FUNCTION_BLOCK FB_FIFO_1 EXTENDS FB_FIFO_OOP
VAR_INPUT
END_VAR
VAR_OUTPUT
END_VAR
VAR
END_VAR

PROPERTY ifEmptyRegister : IF_EmptyRegister
GET
ifEmptyRegister:=super^;
END_GET
END_PROPERTY

PROPERTY ifFillRegister : IF_FillRegister
GET
ifFillRegister:=super^;
END_GET
END_PROPERTY

PROPERTY ifRegister : IF_Register
GET
ifRegister:=super^;
END_GET
END_PROPERTY

END_FUNCTION_BLOCK

(* stored: Version 1.1.0.1
   POU FB_FIFO_1: Id {7d20f1f5-68f8-4dda-a4fa-66e225c03a6c}, SpecialFunc None
   Property ifEmptyRegister: Id {7cd02d5f-3e9f-42f9-b54d-32ee951b56ff}
   Get Get: Id {1e8b9ca5-eaab-40e5-82b7-e5efa8257c99}
   Property ifFillRegister: Id {8fb8c73f-19e7-4556-8ab8-037dd6c98bb0}
   Get Get: Id {175851d4-34ba-4134-ae81-0a0322ea8ba1}
   Property ifRegister: Id {c5d872c1-d02f-454a-8489-bd087fce09c9}
   Get Get: Id {8ccf3126-6346-4196-9f97-54ab605e0003} *)
